// TIA Portal project "R_S_Multi" (V15)

(* hardware
DEVICE "S7-1200 station_1"  S7-1200 Station
   slot 0: "Rack_0"  S7-1200 Rack  Rack  V1.0
   slot 1: "PLC_1"  CPU 1214C DC/DC/Rly  6ES7 214-1HG40-0XB0  V4.0
*)

// ===== PLC "PLC_1"  CPU 1214C DC/DC/Rly =====

VAR_GLOBAL   // PLC tag table "默认变量表"
   "System_Byte" AT %MB1 : Byte;
   "FirstScan" AT %M1.0 : Bool;
   "DiagStatusUpdate" AT %M1.1 : Bool;
   "AlwaysTRUE" AT %M1.2 : Bool;
   "AlwaysFALSE" AT %M1.3 : Bool;
   "Clock_Byte" AT %MB0 : Byte;
   "Clock_10Hz" AT %M0.0 : Bool;
   "Clock_5Hz" AT %M0.1 : Bool;
   "Clock_2.5Hz" AT %M0.2 : Bool;
   "Clock_2Hz" AT %M0.3 : Bool;
   "Clock_1.25Hz" AT %M0.4 : Bool;
   "Clock_1Hz" AT %M0.5 : Bool;
   "Clock_0.625Hz" AT %M0.6 : Bool;
   "Clock_0.5Hz" AT %M0.7 : Bool;
END_VAR

DATA_BLOCK "数据块_1"   // DB5
{ S7_Optimized_Access := 'TRUE' }
VERSION : 0.1
   VAR
      Rec : Array[0..1] of Char;
      Send : Array[0..1] of Byte;
   END_VAR
BEGIN
   Send[0] := 16#0;
END_DATA_BLOCK

DATA_BLOCK "数据块_2"   // DB6
{ S7_Optimized_Access := 'TRUE' }
VERSION : 0.1
   VAR
      Rec : Array[0..1] of Char;
      Send : Array[0..1] of Byte;
   END_VAR
BEGIN
END_DATA_BLOCK

// folder: System blocks/Program resources

DATA_BLOCK "PLC_1_Send_DB"   // DB7
{ S7_Optimized_Access := 'TRUE' }
AUTHOR : SIMATIC
FAMILY : MC7Plus
NAME : TCON_Prm
VERSION : 1.0
// stored: InstanceOfName TCON_Param
"TCON_Param"
BEGIN
   ID := 1;
   REM_TSAP_ID_LEN := 0;
   LOCAL_TSAP_ID[1] := B#16#17;
   LOCAL_TSAP_ID[2] := B#16#70;
   LOCAL_TSAP_ID_LEN := 2;
   ACTIVE_EST := false;
   REM_STADDR[1] := 192;
   REM_STADDR[2] := 168;
   REM_STADDR[4] := 241;
END_DATA_BLOCK

DATA_BLOCK "PLC_1_Send_DB_1"   // DB8
{ S7_Optimized_Access := 'TRUE' }
AUTHOR : SIMATIC
FAMILY : MC7Plus
NAME : TCON_Prm
VERSION : 1.0
// stored: InstanceOfName TCON_Param
"TCON_Param"
BEGIN
   ID := 2;
   REM_TSAP_ID_LEN := 0;
   LOCAL_TSAP_ID[1] := B#16#1B;
   LOCAL_TSAP_ID[2] := B#16#58;
   LOCAL_TSAP_ID_LEN := 2;
   ACTIVE_EST := false;
   REM_STADDR[1] := 192;
   REM_STADDR[2] := 168;
   REM_STADDR[4] := 241;
END_DATA_BLOCK

// folder: (top level)

ORGANIZATION_BLOCK "Main"   // OB1, LAD, ProgramCycle
TITLE = "Main Program Sweep (Cycle)"
{ S7_Optimized_Access := 'TRUE' }
VERSION : 0.1
   VAR_INPUT
      Initial_Call : Bool;   // Initial call of this OB
      Remanence : Bool;   // =True, if remanent data are available
   END_VAR
BEGIN

REGION Network 1
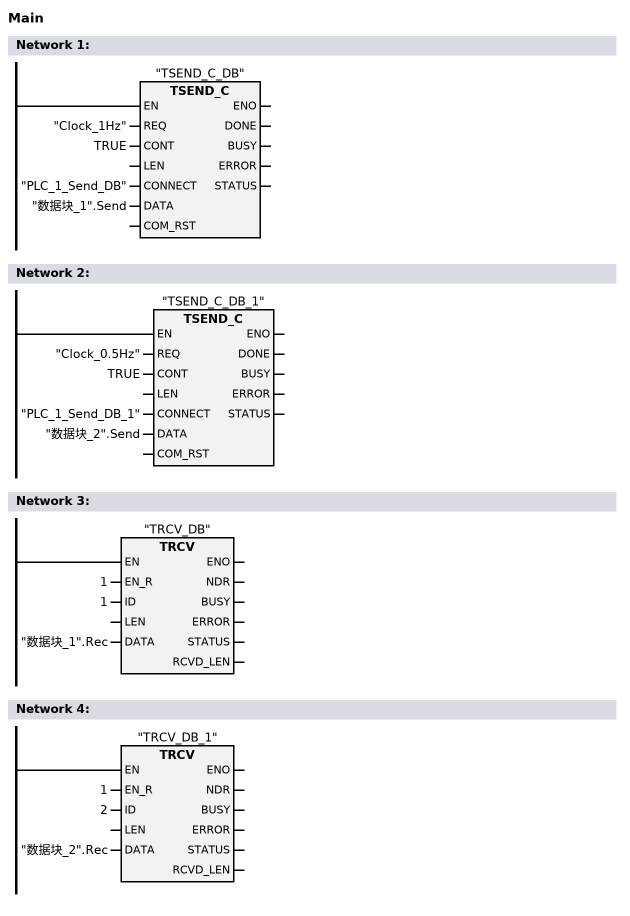
   "TSEND_C_DB"(REQ := "Clock_1Hz", CONT := TRUE, CONNECT := "PLC_1_Send_DB", DATA := "数据块_1".Send);   // TSEND_C
END_REGION

REGION Network 2
   "TSEND_C_DB_1"(REQ := "Clock_0.5Hz", CONT := TRUE, CONNECT := "PLC_1_Send_DB_1", DATA := "数据块_2".Send);   // TSEND_C
END_REGION

REGION Network 3
   "TRCV_DB"(EN_R := 1, ID := 1, DATA := "数据块_1".Rec);   // TRCV
END_REGION

REGION Network 4
   "TRCV_DB_1"(EN_R := 1, ID := 2, DATA := "数据块_2".Rec);   // TRCV
END_REGION
END_ORGANIZATION_BLOCK